Yaskawa INFORM job: shotblast_planes_program.JBI

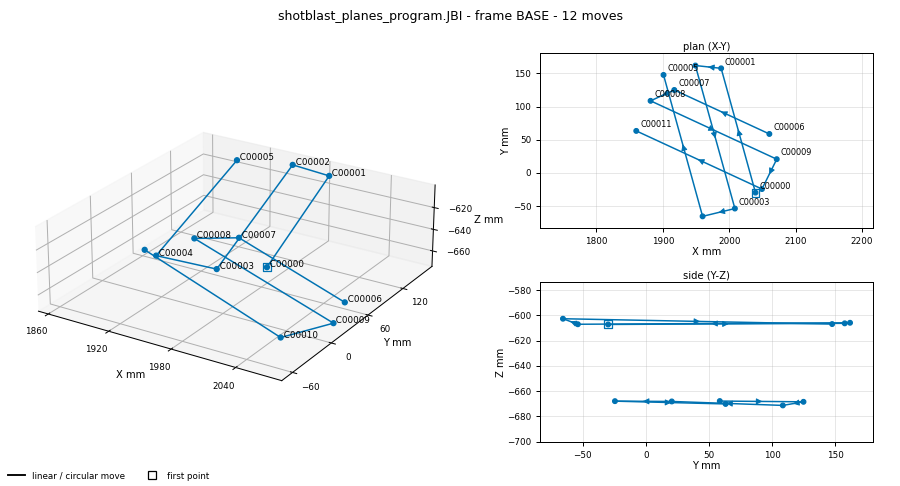
[picture p0: tool path of shotblast_planes_program.JBI in frame BASE, 12 of 15 moves have a stored position in this frame; points joined in program order, loops and branches not executed]
/JOB
//NAME shotblast_planes_program
//POS
///NPOS 12,0,12,0,0,0
///TOOL 0
///POSTYPE BASE
///RECTAN
///RCONF 0,0,0,0,0,0,0,0,0,0,0,0,0,0,0,0,0,0,0,0,0,0,0,0
C00000=2039.650705,-29.739888,-607.131450,175.000000,-5.000000,5.000000
C00001=1987.916717,157.547004,-606.250439,175.000000,-5.000000,5.000000
C00002=1949.081626,161.765561,-605.802439,175.000000,-5.000000,5.000000
C00003=2008.608877,-53.734424,-606.973439,175.000000,-5.000000,5.000000
C00004=1959.955134,-65.518364,-602.600439,175.000000,-5.000000,5.000000
C00005=1901.090291,147.583578,-606.816439,175.000000,-5.000000,5.000000
C00006=2060.557330,58.647147,-667.789300,175.000000,-5.000000,5.000000
C00007=1917.304209,124.909854,-668.373280,175.000000,-5.000000,5.000000
C00008=1881.565992,108.563157,-671.229280,175.000000,-5.000000,5.000000
C00009=2071.686824,20.621471,-668.096280,175.000000,-5.000000,5.000000
C00010=2049.400267,-24.363462,-667.859280,175.000000,-5.000000,5.000000
C00011=1859.991789,63.248720,-670.066280,175.000000,-5.000000,5.000000
///POSTYPE PULSE
///PULSE
EC00000=15360.0
EC00001=15360.0
EC00002=15360.0
EC00003=15360.0
EC00004=15360.0
EC00005=15360.0
EC00006=66560.0
EC00007=66560.0
EC00008=66560.0
EC00009=66560.0
EC00010=66560.0
EC00011=66560.0
//INST
///DATE 2023/08/16 11:59
///ATTR SC,RW,RJ
////FRAME BASE
///GROUP1 RB1,ST1
NOP
MOVJ P009 EX000 VJ=15.00
MOVJ C00000 EC00000 VJ=15.0
CALL JOB:SPYON
MOVL C00001 EC00001 V=150.0
MOVL C00002 EC00002 V=150.0
MOVL C00003 EC00003 V=150.0
MOVL C00004 EC00004 V=150.0
MOVL C00005 EC00005 V=150.0
CALL JOB:SPYOF
MOVJ P009 VJ=15.00
MOVJ C00006 EC00006 VJ=15.0
CALL JOB:SPYON
MOVL C00007 EC00007 V=150.0
MOVL C00008 EC00008 V=150.0
MOVL C00009 EC00009 V=150.0
MOVL C00010 EC00010 V=150.0
MOVL C00011 EC00011 V=150.0
CALL JOB:SPYOF
MOVJ P009 VJ=15.00
END
